{attribute 'linkalways'} 
{attribute 'no_explicit_call' := 'This FB is a CLASS and must be accessed using methods or properties'}
{attribute 'enable_dynamic_creation'}
FUNCTION_BLOCK _ETcVnCodeType EXTENDS EnumDatatypeBase
VAR
	localData : ETcVnCodeType;
	activeData : REFERENCE TO ETcVnCodeType;
	enumBaseDatatype : _ULINT(localData);
END_VAR

METHOD PRIVATE AddLocalEnumeration
VAR_INPUT
	Enumeration : T_MAXSTRING;
	Value : ETcVnCodeType;
END_VAR
AddEnumeration(Enumeration, Value);
END_METHOD

PROPERTY PUBLIC Address : PVOID
GET
Address := ADR(activeData);
END_GET
END_PROPERTY

METHOD PUBLIC ClearReference
VAR_INPUT
END_VAR
activeData REF= localData;
SetBaseDatatypeReference();
END_METHOD

METHOD PUBLIC Clone : I_Datatype
VAR
    pClone : POINTER TO _ETcVnCodeType;
END_VAR
pClone := __NEW(_ETcVnCodeType(InitialValue := Value));
Clone := pClone^;
END_METHOD

METHOD FB_init : BOOL
VAR_INPUT
	bInitRetains : BOOL; // if TRUE, the retain variables are initialized (warm start / cold start)
	bInCopyCode : BOOL;  // if TRUE, the instance afterwards gets moved into the copy code (online change)
	InitialValue : ETcVnCodeType;
END_VAR
localData := InitialValue;
AddBaseDatatype(enumBaseDatatype);
ClearReference();

AddLocalEnumeration('TCVN_CT_ANY', ETcVnCodeType.TCVN_CT_ANY);
AddLocalEnumeration('TCVN_CT_1D', ETcVnCodeType.TCVN_CT_1D);
AddLocalEnumeration('TCVN_CT_2D', ETcVnCodeType.TCVN_CT_2D);
AddLocalEnumeration('TCVN_CT_QR', ETcVnCodeType.TCVN_CT_QR);
AddLocalEnumeration('TCVN_CT_DATAMATRIX', ETcVnCodeType.TCVN_CT_DATAMATRIX);
AddLocalEnumeration('TCVN_CT_DOTCODE', ETcVnCodeType.TCVN_CT_DOTCODE);
END_METHOD

PROPERTY PUBLIC Identifier : T_MAXSTRING
GET
Identifier := 'ETcVnCodeType';
END_GET
END_PROPERTY

METHOD IsEnumeratorValueEqual : BOOL
VAR_INPUT
	Enumerator : I_KeyValueForwardEnumerator;
END_VAR
VAR
	storedValue : ETcVnCodeType;
END_VAR
IF NOT Enumerator.TryGet(storedValue) THEN
	RETURN;
END_IF

IsEnumeratorValueEqual := storedValue = activeData;
END_METHOD

METHOD PUBLIC MakeReferenceTo
VAR_INPUT
	ReferenceTarget : REFERENCE TO ETcVnCodeType;
END_VAR
activeData REF= ReferenceTarget;
SetBaseDatatypeReference();
END_METHOD

METHOD PROTECTED SetBaseDatatypeReference
VAR_INPUT
END_VAR
enumBaseDatatype.MakeReferenceTo(activeData);
END_METHOD

PROPERTY PUBLIC Size : UDINT
GET
Size := SIZEOF(activeData);
END_GET
END_PROPERTY

METHOD TryMakeReferenceTo : BOOL
VAR_INPUT
	Target : I_Datatype;
END_VAR
VAR
	pTargetData : POINTER TO ETcVnCodeType;
END_VAR
IF NOT IsEquivalentTo(Target) THEN
	RETURN;
END_IF

pTargetData := Target.Address;
activeData REF= pTargetData^;
SetBaseDatatypeReference();
TryMakeReferenceTo := TRUE;
END_METHOD

PROPERTY PUBLIC Value : ETcVnCodeType
GET
Value := activeData;
END_GET
SET
activeData := Value;
END_SET
END_PROPERTY

END_FUNCTION_BLOCK

(* stored: Version 1.1.0.1, ProductVersion 3.1.4026.18
   POU _ETcVnCodeType: Id {54809282-376a-0b1a-0e16-380091fac695}, SpecialFunc None
   Folder Core: Id {80368904-e50d-0768-2ba2-9f7c1a4a1cb0}
   Folder Protected: Id {2649b9e1-f0ea-0f58-0d7c-db049f8f9eaf}
   Folder Customize: Id {8d3de4b2-caa4-0bd9-2911-bb194ca677fa}
   Folder Constructor: Id {54a2529a-dfb6-08fb-0d90-dfe9bb88471a}
   Folder Private: Id {0bef58f8-bb09-0a87-26e6-4314e13986f4}
   Folder Protected: Id {96151ad0-c95a-0174-0653-7973f6cb59e7}
   Method AddLocalEnumeration: Id {691fea77-9867-0d96-345b-fc633e28cdbe}
   Property Address: Id {0f18952f-4bd0-0002-277c-be4136624bba}
   Get Get: Id {3f4e3766-370d-090b-22b2-41fd22afc24b}
   Method ClearReference: Id {6953848d-df01-0834-127d-c4a737974180}
   Method Clone: Id {312a2d32-0422-09d3-3a48-9874d3b2d600}
   Method FB_init: Id {5fac7567-2741-0954-152d-b158cb48c629}
   Property Identifier: Id {9b6242fb-d1e3-0a34-389e-121225c34765}
   Get Get: Id {41c38992-6a1e-0b69-2d68-6f06c206291e}
   Method IsEnumeratorValueEqual: Id {3e6efbd2-e1bc-0b6f-387f-39bd29688a5c}
   Method MakeReferenceTo: Id {8ebbae99-c367-06fa-30fa-c062cadb369c}
   Method SetBaseDatatypeReference: Id {a4f8a584-aca7-0a40-2831-1dfafa3c277a}
   Property Size: Id {76f92abe-99a2-0586-174c-977a691708b7}
   Get Get: Id {c390a662-9830-08e7-2318-6edc2abfd142}
   Method TryMakeReferenceTo: Id {b635687a-af63-0da3-23df-4a824f0b04ab}
   Property Value: Id {60e4c4d1-f29e-054d-2ca2-f48a37c8ec94}
   Get Get: Id {d45ab43a-f878-09dc-30a3-c39f9b6aad82}
   Set Set: Id {df042a17-5240-013b-0324-b6adf9a5a599} *)
